// TIA Portal V20 export
DATA_BLOCK "SP203"   // DB314
// stored: MemoryReserve 100
   VAR
      "MAIN OP MODE SLELECT SS.AUTO" : Bool;
      "MAIN OP HOME PBL (GREEN)" : Bool;
      "MAIN OP SAFETY RESET PBL (BLUE)" : Bool;
      "MAIN OP SCS MODE SLELECT SS.AUTO" : Bool;
      "MAIN OP MODE SLELECT SS.MANUAL" : Bool;
      "MAIN OP ENABLE PBL (WHITE)" : Bool;
      "MAIN OP SCS MODE SLELECT SS.SETUP" : Bool;
      "MAIN OP SCS MODE SLELECT SS.DISABLE" : Bool;
   END_VAR
BEGIN
END_DATA_BLOCK
